(* IEC 61131-3 sources: repolevel_ST_code_completion/output/0121完整版本/repoeval_Builder_Application_RPI/readful_result_no_provide, 5 files *)

(* ---- Director.st ---- *)
{attribute 'enable_dynamic_creation'}
//The director class is responsible to delegate the construction of the final product object
// to a concrete builder object.
FUNCTION_BLOCK Director
VAR_INPUT
  //Reference to the builder that is going to be building the final product object.
  inputConcreteBuilder : ConcreteBuilder;
END_VAR
VAR_OUTPUT
END_VAR
VAR
  //Holds a reference to the concrete builder object to send the specifications of the final product to it.
  concreteBuilder : ConcreteBuilder;
END_VAR

// Stores the reference to the builder object in the field `concreteBuilder`
concreteBuilder := inputConcreteBuilder;

//The Director tells its concreteBuilder instance to build the final product step by step passing the specifications stored in the
// concreteBuilder array THIS^.specifications[1..4]

//Step 1 "Main Part"
concreteBuilder.Set_Main_Part(concreteBuilder.specifications[1]);
//Step 2 "Part 1"
concreteBuilder.Set_Part1(concreteBuilder.specifications[2]);
//Step 3 "Part 2"
concreteBuilder.Set_Part2(concreteBuilder.specifications[3]);
//Step 4 "Part 3"
concreteBuilder.Set_Part3(concreteBuilder.specifications[4]);

// The final product object should be processed, ensure its proper usage
concreteBuilder.Get_Result(); // This call must be further managed by the application
END_FUNCTION_BLOCK

(* ---- ConcreteBuilder.st ---- *)
VAR
    // Holds an internal reference to how the final product should be so the builder class can build it on the fly
    // without any help from other classes excepting the Director class that is going to be passing the special
    // specifications to the builder.
    localProduct : Product;

    // Stores the specifications, sent by the client, of the final product to be built.
    specifications : ARRAY [1..4] OF STRING;
END_VAR

// Sets the main part of the product based on the specification
METHOD Set_Main_Part : BOOL
VAR_INPUT
  mainPartSpec : STRING;
END_VAR
localProduct.MainPart := mainPartSpec;
RETURN; // Ends execution with a return value if needed

// Sets the first part of the product based on the specification
METHOD Set_Part1
VAR_INPUT
    part1Spec : STRING;
END_VAR
VAR_OUTPUT
END_VAR
VAR
END_VAR
localProduct.Part1 := part1Spec;

// Sets the second part of the product based on the specification
METHOD Set_Part2
VAR_INPUT
    part2Spec : STRING;
END_VAR
VAR_OUTPUT
END_VAR
VAR
END_VAR
localProduct.Part2 := part2Spec;

// Sets the third part of the product based on the specification
METHOD Set_Part3
VAR_INPUT
    part3Spec : STRING;
END_VAR
VAR_OUTPUT
END_VAR
VAR
END_VAR
localProduct.Part3 := part3Spec;
END_FUNCTION_BLOCK

(* ---- Director_Construct.st ---- *)
VAR
	//Holds a reference to the concrete builder object to send the specifications of the final product to it.
	concreteBuilder : ConcreteBuilder(specs := THIS^.inputConcreteBuilder.specifications);
END_VAR

//Step 1 "Main Part"
concreteBuilder.Set_Main_Part(concreteBuilder.specifications[1]);
//Step 2 "Part 1"
concreteBuilder.Set_Part1(concreteBuilder.specifications[2]);
//Step 3 "Part 2"
concreteBuilder.Set_Part2(concreteBuilder.specifications[3]);
//Step 4 "Part 3"
concreteBuilder.Set_Part3(concreteBuilder.specifications[4]);

//Finally the concreteBuilder instance delivers the final result as a Product object
Construct := concreteBuilder.Get_Result();
RETURN;
END_OTHER

(* ---- Product.st ---- *)
VAR
    // Temporary variable to hold the dynamically created product
// Index variable for iterating through specifications
  i : INT;
END_VAR

// Initialize the existing product fields directly without using tempProduct
mainPart := '';
part1 := '';
part2 := '';
part3 := '';

// Manually assign or override the product inputs if necessary based on existing logic
// For example, inputs may already provide sufficient data

// Use the existing input variables as-is without creating temporary objects
END_FUNCTION_BLOCK

(* ---- Product_toString.st ---- *)
VAR
    tempString: STRING;
END_VAR

tempString := CONCAT(mainPart, part1);
tempString := CONCAT(tempString, part2);
tempString := CONCAT(tempString, part3);
toString := tempString;
RETURN;
END_OTHER
